TYPE ST_FireDetectionSet :
STRUCT
	b_SilenceSounder	:	BOOL; //only disables currently activated alarm.
	b_TestSounder		:	BOOL;
END_STRUCT
END_TYPE

(* stored: Version 1.1.0.1, ProductVersion 3.1.4024.12
   DUT ST_FireDetectionSet: Id {5cb45d6d-8880-457c-8f25-162a610efcce} *)
